(* IEC 61131-3 sources: Industry-PLC-LLM/data/PLCBEAD_repo/PLCBEAD_PLCEmbed-main/PLC-BEAD/Source/GEB/REAL_TO_FRAC, 1 file *)

(* ---- REAL_TO_FRAC.ST ---- *)
TYPE oscat_FRACTION :
	STRUCT
		NUMERATOR : INT;
		DENOMINATOR : INT;
	END_STRUCT;
END_TYPE

FUNCTION_BLOCK REAL_TO_FRAC_Block

	VAR_INPUT
		X :	REAL;
		N :	INT;
	END_VAR

	VAR_OUTPUT
		REAL_TO_FRAC :	oscat_FRACTION;
	END_VAR

	VAR
		temp :	DINT;
		SIGN :	BOOL;
		X_gerundet :	DINT;
		X_ohne_Nachkomma :	REAL;
		Numerator :	DINT := 1;
		Denominator :	DINT := 0;
		Numerator_old :	DINT := 0;
		Denominator_old :	DINT := 1;
	END_VAR

	IF X < 0.0 THEN
		SIGN := TRUE;								(* Vorzeichen merken *)
		X := ABS(X);								(* Absolutwert berechnen *)
	END_IF;

	REPEAT
		X_gerundet := REAL_TO_DINT(X);

		temp := numerator * X_gerundet + numerator_old;		(* Zaehler um Vorkammawert erweitern *)
		numerator_old := numerator;							(* Zaehler der letzten Berechnung speichern *)
		numerator := temp;									(* Zaehler dieser Berechnung speichern *)

		temp := denominator * X_gerundet + denominator_old;	(* Nenner um Vorkammawert erweitern *)
		denominator_old := denominator;						(* Nenner der letzten Berechnung speichern *)
		denominator := temp;								(* Nenner dieser Berechnung speichern *)

		X_ohne_Nachkomma := DINT_TO_REAL(X_gerundet);
		IF X = X_ohne_Nachkomma THEN						(* Bruch geht ohne Rest auf *)
			IF ABS(denominator) <= INT_TO_DINT(N) THEN		(* keIN Rundungsfehler *)
				numerator_old := numerator;					(* Numerator_old wird von Funktion zur�ckgegeben *)
				denominator_old := denominator;				(* Denominator_old wird von Funktion zur�ckgegeben *)
			END_IF;
			EXIT;											(* keine weitere Berechnung notwendig *)
		ELSE
			X := 1.0 / (X - X_ohne_Nachkomma);				(* Kehrwert vom Rest -> Neuer Bruch *)
		END_IF;

	UNTIL
		( ABS(Denominator) > INT_TO_DINT(N))
	END_REPEAT;

	IF SIGN THEN
		REAL_TO_FRAC.NUMERATOR := -1 * ABS(DINT_TO_INT(numerator_old));
	ELSE
		REAL_TO_FRAC.NUMERATOR :=  ABS(DINT_TO_INT(numerator_old));
	END_IF;

	REAL_TO_FRAC.DENOMINATOR := ABS(DINT_TO_INT(denominator_old));

END_FUNCTION_BLOCK

PROGRAM program0

	VAR
		X :	REAL;
		N :	INT;

        REAL_TO_FRAC :	oscat_FRACTION;
		func_block : REAL_TO_FRAC_Block;
	END_VAR
		func_block.X := X;
		func_block.N := N;
		func_block();
		REAL_TO_FRAC := func_block.REAL_TO_FRAC;

END_PROGRAM
